(*******************************************************************************
                          protoc-gen-twincat V0.0.0.0                           
                  https://github.com/TcHaxx/protoc-gen-twincat                  
*******************************************************************************)
{attribute 'qualified_only'}
{attribute 'strict'}
{attribute 'to_string'}
TYPE E_DataType :
(
	DATA_TYPE_UNKNOWN := 0,
	DATA_TYPE_TEMPERATURE := 1,
	DATA_TYPE_PRESSURE := 2,
	DATA_TYPE_HUMIDITY := 3
) BYTE;
END_TYPE

(* stored: Version 1.1.0.1
   DUT E_DataType: Id 1be0b3be-aa6c-4d93-81f7-f74b2a6cc4ac *)
